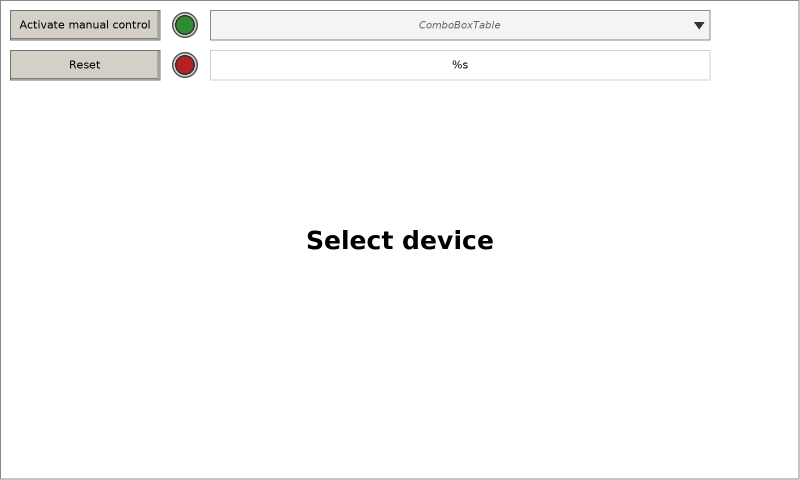
VISUALIZATION ManualControl  // 800x480
VAR_IN_OUT
	fbManualControler	: FB_ManualController ;
	
END_VAR
    Frame (0,0 800x480), input disabled if: fbManualControler.bDisableManualInputs, frame switch variable: fbManualControler.eDevType
        shows VisuUndefinedControl()
        shows VisuValveControl(fbManualControler := fbManualControler)
        shows VisuCylinderControl(fbManualControler := fbManualControler)
        shows VisuAxisControl(fbManualControler := fbManualControler)
        shows VisuPushbuttonLightControl(fbManualControler := fbManualControler)
        shows VisuDigitalInputControl(fbManualControler := fbManualControler)
        shows VisuAnlogInputControl(fbManualControler := fbManualControler)
        shows VisuDigitalOutControl(fbManualControler := fbManualControler)
        shows VisuAnalogOutControl(fbManualControler := fbManualControler)
        shows VisuPWMControl(fbManualControler := fbManualControler)
        shows VisuDoublePWMControl(fbManualControler := fbManualControler)
        shows VisuEncoderInput(fbManualControler := fbManualControler)
        shows VisuAnalogAxisControl(fbManualControler := fbManualControler)
        shows VisuTwoVelocityAxisControl(fbManualControler := fbManualControler)
        shows VisuKL5151Control(fbManualControler := fbManualControler)
        shows VisuKL15XXControl(fbManualControler := fbManualControler)
    Button (10,10 150x30), "Activate manual control", pressed state: fbManualControler.bManualActive
        toggle fbManualControler.bManualActive
    Lamp1 (170,50 30x30), tooltip "component fault active", variable: fbManualControler.bErroractive, style: Lamp-Lamp1-Red
    Lamp1 (170,10 30x30), tooltip "Manual control active", variable: fbManualControler.bManual, style: Lamp-Lamp1-Green
    Textfield (210,50 500x30), "%s", text variable: fbManualControler.sDeviceState
    Button (10,50 150x30), "Reset"
        tap fbManualControler.bReset
    ComboBoxTable (210,10 500x30), variable: fbManualControler.nCmdLookupindex, data array: fbManualControler.arDeviceArray
        p1128707560: fbManualControler.nNumberOfDevices
        p3854506369: fbManualControler.arDeviceArray[INDEX].sName
        p1892666644: fbManualControler.arDeviceArray[INDEX].sType
        p338671338: fbManualControler.arDeviceArray[INDEX].pFunction^
END_VISUALIZATION

// ---- Screens/Manual/toManualButton.TcVIS
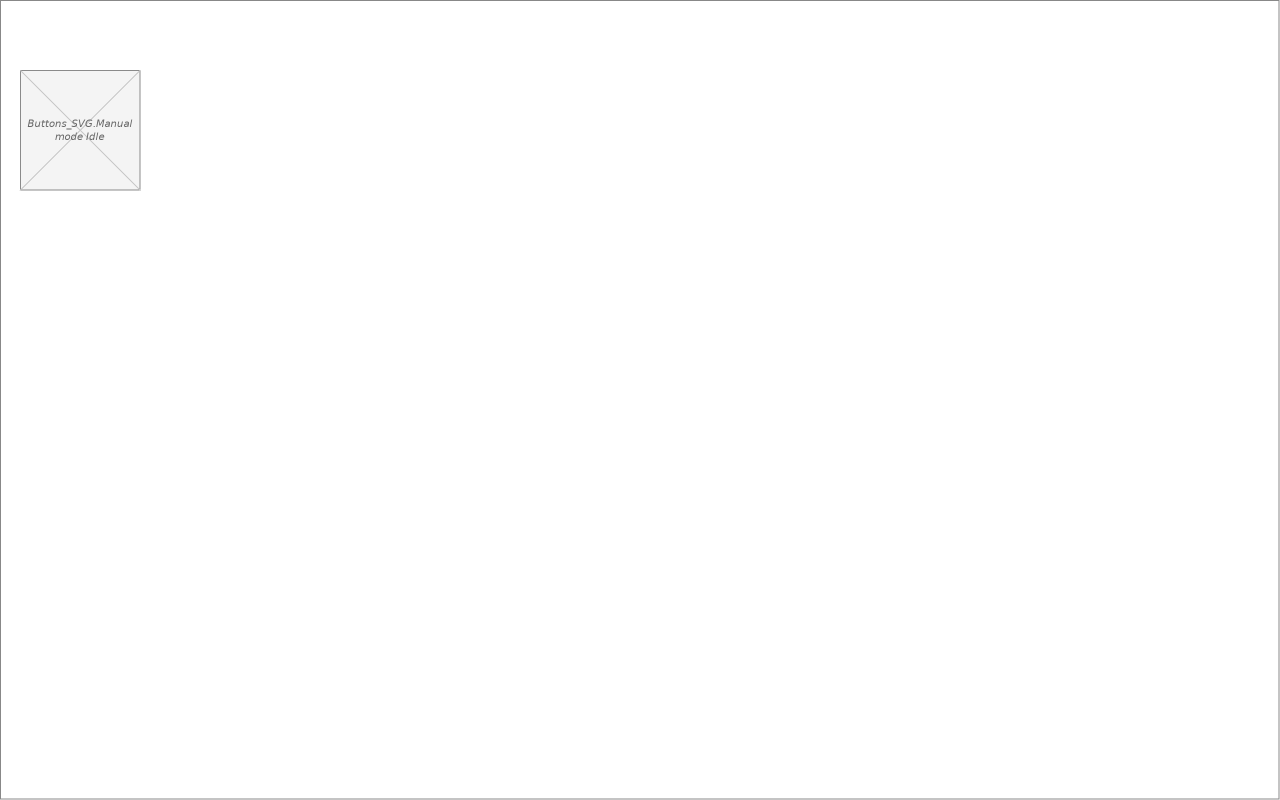
VISUALIZATION toManualButton  // 1280x800
    Image (20,70 120x120), image: Buttons_SVG.Manual mode Idle
        OnMouseClick: toggle GVL_HMI.bCmdManual
END_VISUALIZATION

// ---- Screens/Parameter/ParameterControl.TcVIS
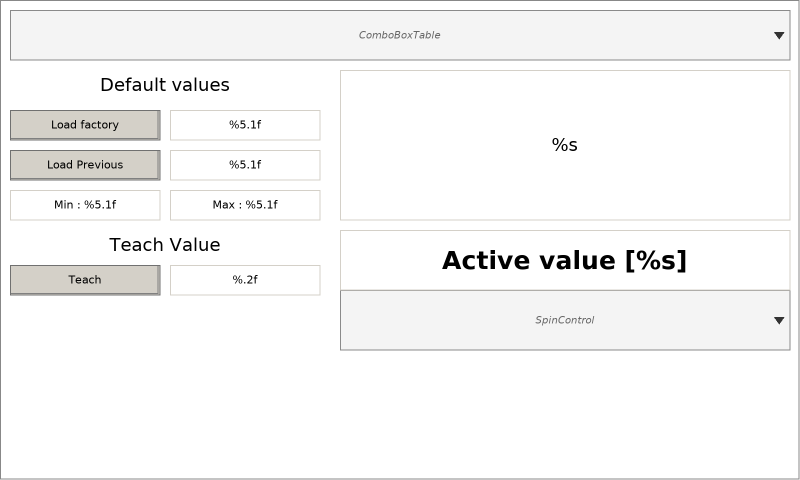
VISUALIZATION ParameterControl  // 800x480
    ComboBoxTable (10,10 780x50), variable: GVL_Parameters.fbParameterHandler.nLookupIndex, data array: GVL_Parameters.fbParameterHandler.arParameters
        p1128707560: GVL_Parameters.fbParameterHandler.nNumberOfParameters
        p3854506369: GVL_Parameters.fbParameterHandler.arParameters[INDEX].nNumber
        p1892666644: GVL_Parameters.fbParameterHandler.arParameters[INDEX].sName
        p338671338: GVL_Parameters.fbParameterHandler.arParameters[INDEX].sType
        p2170511999: GVL_Parameters.fbParameterHandler.arParameters[INDEX].pParameter^
    Group (10,70 310x150)
        Button (0,40 150x30), "Load factory"
            tap GVL_Parameters.fbParameterHandler.bCmdLoadfactory
        Label (0,0 310x30), "Default values"
        Textfield (160,40 150x30), "%5.1f", text variable: GVL_Parameters.fbParameterHandler.arParameters[GVL_Parameters.fbParameterHandler.nLookupIndex].pParameter^.fFactory
            OnMouseClick: write the text variable via VisuDialogs.Numpad, min GVL_Parameters.fbParameterHandler.arParameters[GVL_Parameters.fbParameterHandler.nLookupIndex].pParameter^.fMinimum, max GVL_Parameters.fbParameterHandler.arParameters[GVL_Parameters.fbParameterHandler.nLookupIndex].pParameter^.fMaximum
        Button (0,80 150x30), "Load Previous"
            tap GVL_Parameters.fbParameterHandler.bCmdLoadFromPrevious
        Textfield (160,80 150x30), "%5.1f", text variable: GVL_Parameters.fbParameterHandler.arParameters[GVL_Parameters.fbParameterHandler.nLookupIndex].pParameter^.fSaved
        Textfield (160,120 150x30), "Max : %5.1f", text variable: GVL_Parameters.fbParameterHandler.arParameters[GVL_Parameters.fbParameterHandler.nLookupIndex].pParameter^.fMaximum
            OnMouseClick: write the text variable via VisuDialogs.Numpad
        Textfield (0,120 150x30), "Min : %5.1f", text variable: GVL_Parameters.fbParameterHandler.arParameters[GVL_Parameters.fbParameterHandler.nLookupIndex].pParameter^.fMinimum
            OnMouseClick: write the text variable via VisuDialogs.Numpad
    Textfield (340,70 450x150), "%s", text variable: GVL_Parameters.fbParameterHandler.arParameters[GVL_Parameters.fbParameterHandler.nLookupIndex].pParameter^.sDiscription
    SpinControl (340,290 450x60), variable: GVL_Parameters.fbParameterHandler.arParameters[GVL_Parameters.fbParameterHandler.nLookupIndex].pParameter^.fValue
        p576042468: GVL_Parameters.fbParameterHandler.arParameters[GVL_Parameters.fbParameterHandler.nLookupIndex].pParameter^.fMinimum
        p651134158: GVL_Parameters.fbParameterHandler.arParameters[GVL_Parameters.fbParameterHandler.nLookupIndex].pParameter^.fMaximum
        OnMouseClick: write the text variable via VisuDialogs.Numpad, min GVL_Parameters.fbParameterHandler.arParameters[GVL_Parameters.fbParameterHandler.nLookupIndex].pParameter^.fMinimum, max GVL_Parameters.fbParameterHandler.arParameters[GVL_Parameters.fbParameterHandler.nLookupIndex].pParameter^.fMaximum
    Textfield (340,230 450x60), "Active value [%s]", text variable: GVL_Parameters.fbParameterHandler.arParameters[GVL_Parameters.fbParameterHandler.nLookupIndex].pParameter^.sUnit
    Group (10,230 310x65)
        Label (0,0 310x30), "Teach Value"
        Textfield (160,35 150x30), "%.2f", text variable: GVL_Parameters.fbParameterHandler.arParameters[GVL_Parameters.fbParameterHandler.nLookupIndex].pParameter^.fPrepared
        Button (0,35 150x30), "Teach"
            tap GVL_Parameters.fbParameterHandler.bCmdAcceptTeach
END_VISUALIZATION

// ---- Screens/Parameter/ParButton_PNG.TcVIS
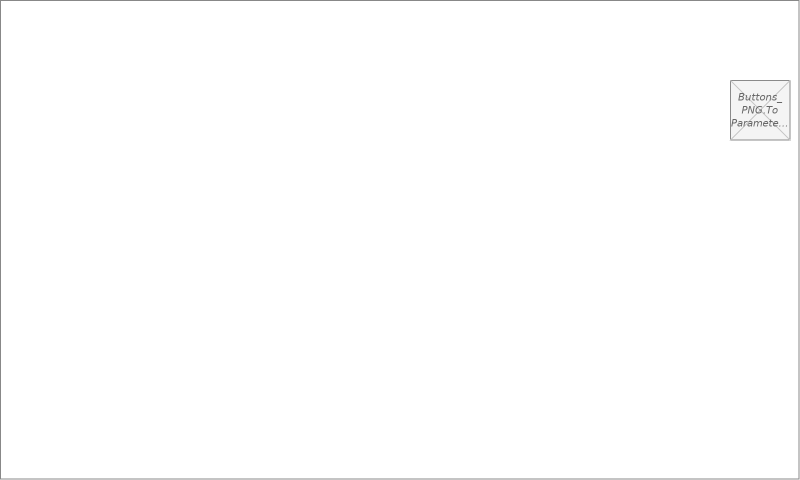
VISUALIZATION ParButton_PNG  // 800x480
VAR_IN_OUT
	bCmdParameter	: BOOL ; // to parameter screen
END_VAR
    Image (730,80 60x60), image: Buttons_PNG.To Parameter Screen
        OnMouseClick: toggle bCmdParameter
END_VISUALIZATION

// ---- Screens/Startup Screen/LogoScreen_PNG.TcVIS
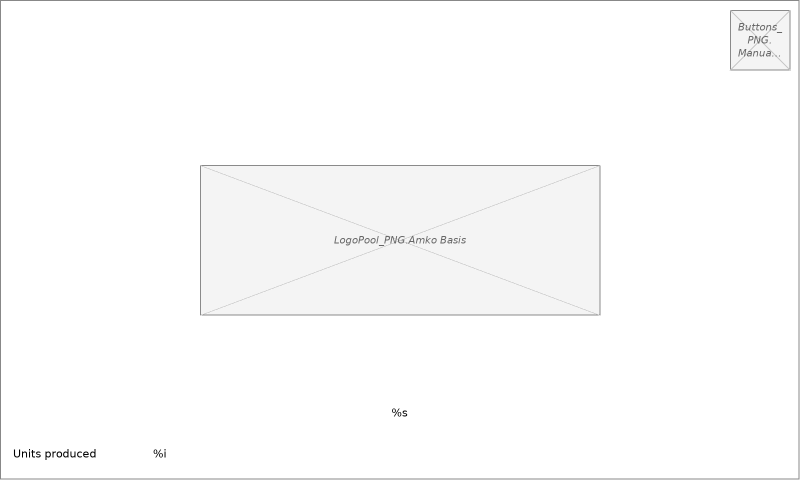
VISUALIZATION LogoScreen_PNG  // 800x480
VAR_INPUT
	nUnitsProduced	: UDINT; // HMI Main total units produced
END_VAR
VAR_IN_OUT
	bCmdManual		: BOOL ; // HMI switch to manual mode
END_VAR
    Frame (0,0 800x480)
        shows ManualButton_PNG(bCmdManual := bCmdManual)
    Image (200,165 400x150), image: LogoPool_PNG.Amko Basis
    Textfield (183,404 433x18), "%s", tooltip "Operator messagages", text variable: GVL_Message.sOPeratorMessage
    Textfield (110,439 100x30), "%i", text variable: nUnitsProduced
    Label (10,439 100x30), "Units produced"
END_VISUALIZATION

// ---- Screens/Startup Screen/LogoScreenBliss_PNG.TcVIS
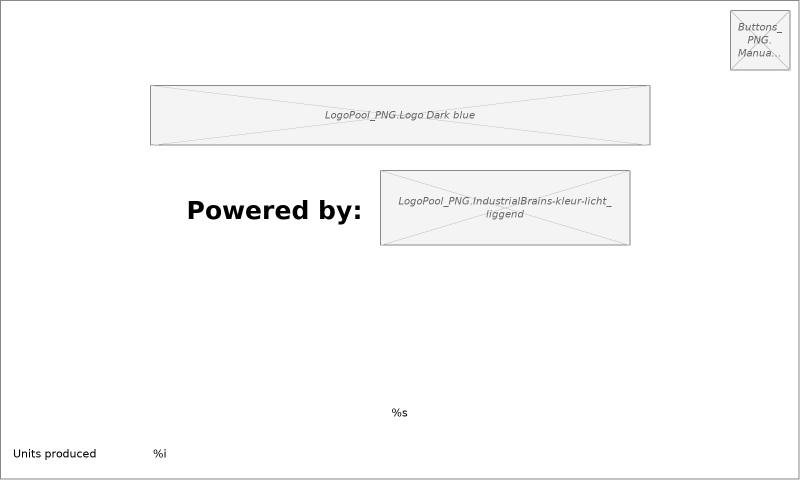
VISUALIZATION LogoScreenBliss_PNG  // 800x480
VAR_INPUT
	nUnitsProduced	: UDINT; // HMI Main total units produced
END_VAR
VAR_IN_OUT
	bCmdManual		: BOOL ; // HMI switch to manual mode
END_VAR
    Frame (0,0 800x480)
        shows ManualButton_PNG(bCmdManual := bCmdManual)
    Image (150,85 500x60), image: LogoPool_PNG.Logo Dark blue
    Image (380,170 250x75), image: LogoPool_PNG.IndustrialBrains-kleur-licht_liggend
    Textfield (183,404 433x18), "%s", tooltip "Operator messagages", text variable: GVL_Message.sOPeratorMessage
    Textfield (110,439 100x30), "%i", text variable: nUnitsProduced
    Label (10,439 100x30), "Units produced"
    Label (179,150 200x120), "Powered by:"
END_VISUALIZATION

// ---- Screens/Startup Screen/LogoScreen_SVG.TcVIS
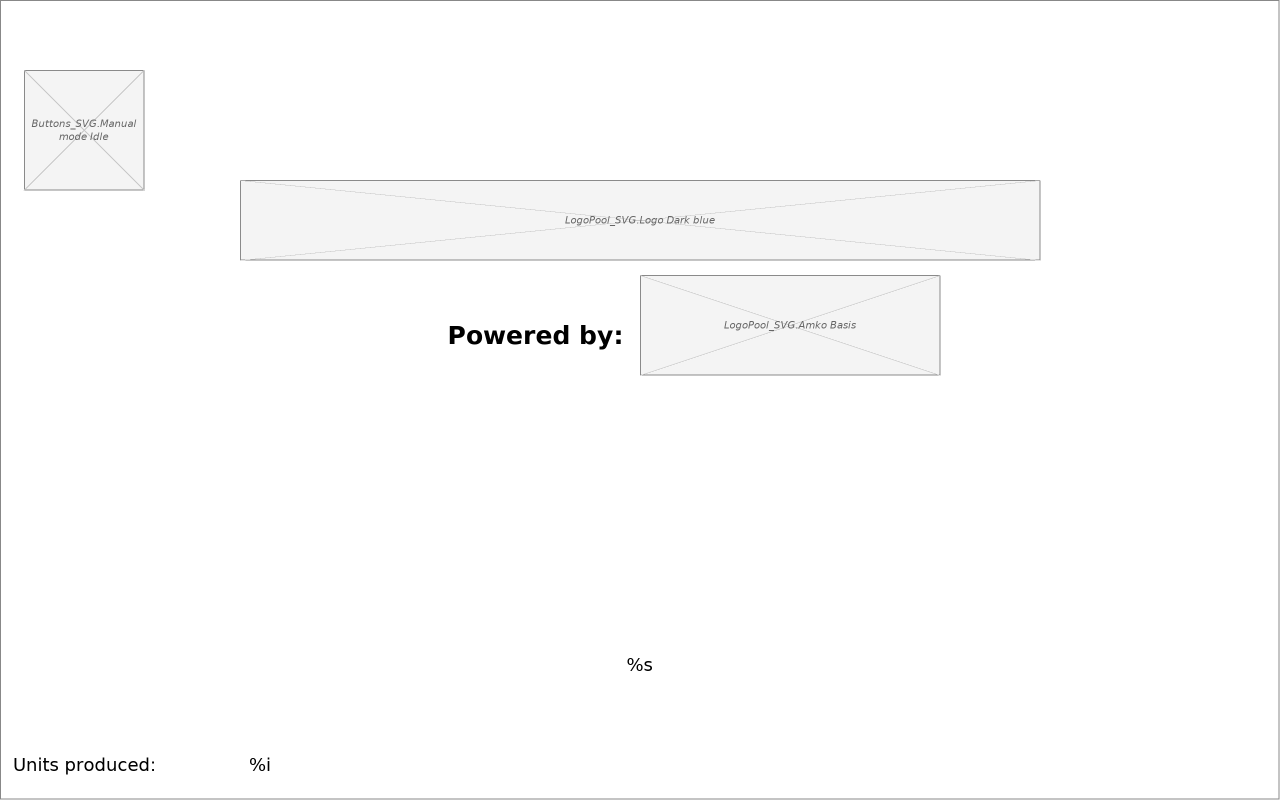
VISUALIZATION LogoScreen_SVG  // 1280x800
VAR_IN_OUT
	nUnitsProduced : UDINT ; // Units produced in machine lifetime
END_VAR
    Frame (4,0 1280x800)
        shows toManualButton()
    Image (240,180 800x80), image: LogoPool_SVG.Logo Dark blue
    Image (640,275 300x100), image: LogoPool_SVG.Amko Basis
    Label (440,275 200x120), "Powered by:"
    Textfield (240,650 800x30), "%s", tooltip "Operator messagages", text variable: GVL_Message.sOPeratorMessage
    Textfield (160,750 200x30), "%i", text variable: nUnitsProduced
    Label (10,750 150x30), "Units produced:"
END_VISUALIZATION

// ---- Screens/Startup Screen/LogoScreenBlanc_SVG.TcVIS
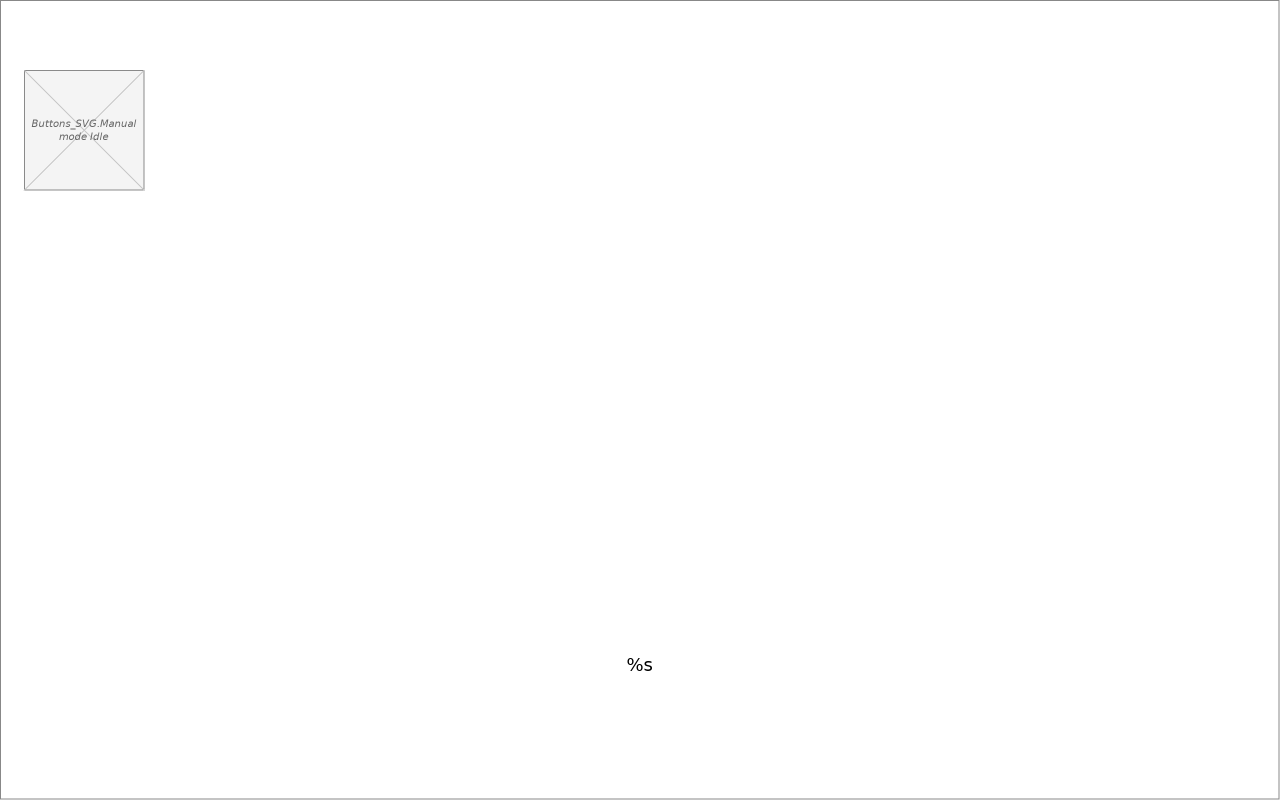
VISUALIZATION LogoScreenBlanc_SVG  // 1280x800
    Frame (4,0 1280x800)
        shows toManualButton()
    Textfield (240,650 800x30), "%s", tooltip "Operator messagages", text variable: GVL_Message.sOPeratorMessage
END_VISUALIZATION

// ---- Screens/State_PNG/Idle_PNG.TcVIS
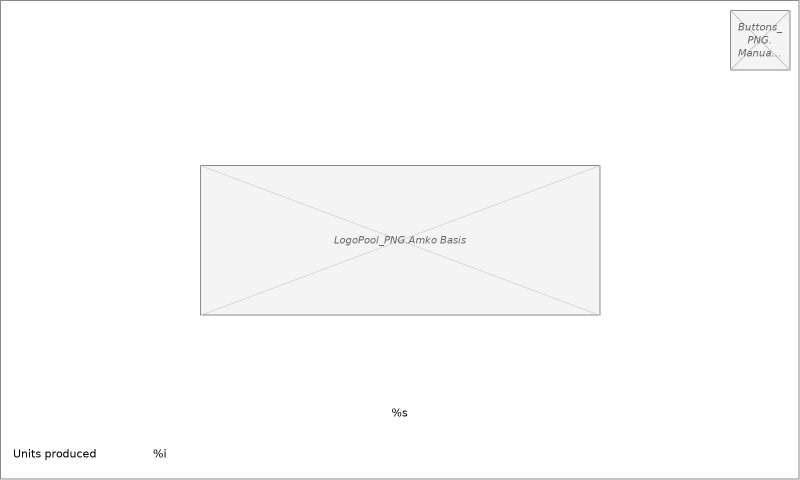
VISUALIZATION Idle_PNG  // 800x480
VAR_IN_OUT
	nUnitsProduced	: UDINT ;
END_VAR
    Frame (0,0 800x480)
        shows LogoScreen_PNG(nUnitsProduced := nUnitsProduced, bCmdManual := GVL_HMI.bCmdManual)
END_VISUALIZATION

// ---- Screens/State_PNG/Manual_PNG.TcVIS
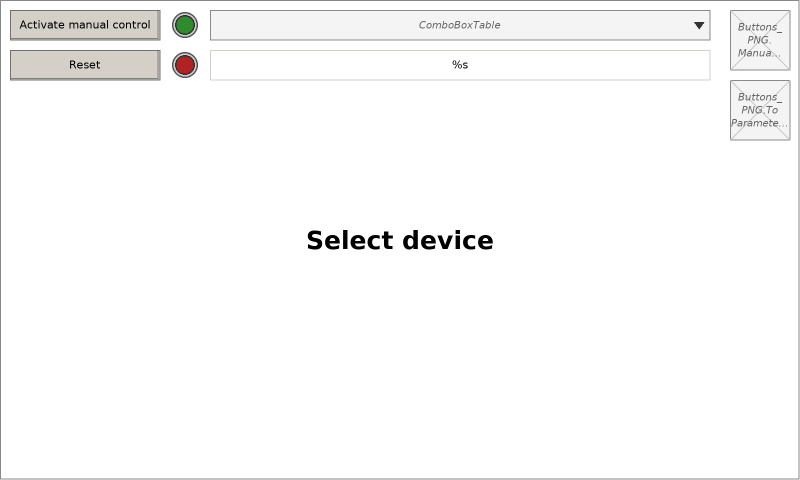
VISUALIZATION Manual_PNG  // 800x480
VAR_IN_OUT
	bCmdManual  	: BOOL ; // switch to manual screen
	bCmdParameter	: BOOL ; // switch to parameter screen
END_VAR
    Frame (0,0 800x480)
        shows ManualControl(fbManualControler := Device_Library.GVL_DevManual.fbManualControler)
    Frame (0,0 800x480)
        shows ManualButton_PNG(bCmdManual := bCmdManual)
    Frame (0,0 800x480)
        shows ParButton_PNG(bCmdParameter := bCmdParameter)
END_VISUALIZATION

// ---- Screens/State_PNG/Parameter_PNG.TcVIS
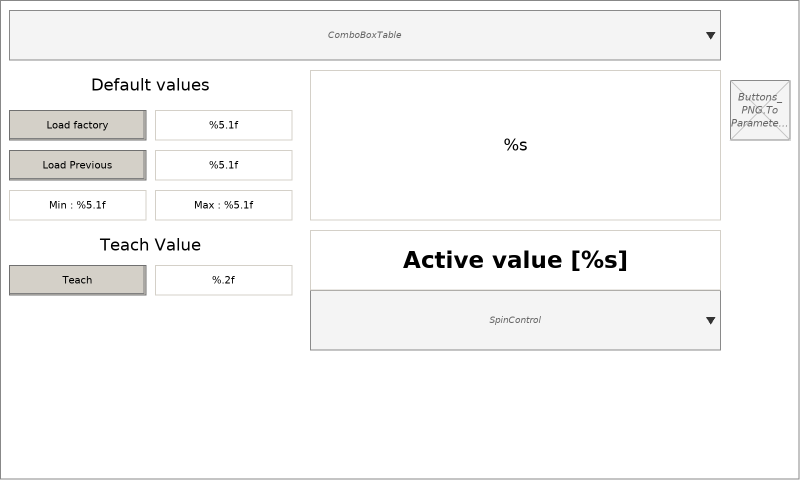
VISUALIZATION Parameter_PNG  // 800x480
VAR_IN_OUT
	bCmdParameter : BOOL ; // Return from parameter screen
END_VAR
    Frame (0,0 800x480)
        shows ParButton_PNG(bCmdParameter := bCmdParameter)
    Frame (0,0 730x480)
        shows ParameterControl()
END_VISUALIZATION

// ---- Screens/State_PNG/Settings_PNG.TcVIS
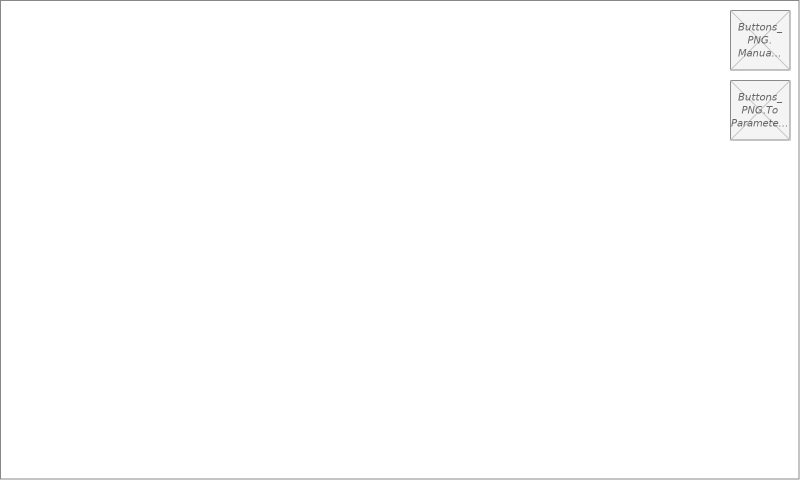
VISUALIZATION Settings_PNG  // 800x480
    Frame (0,0 800x480)
        shows ManualButton_PNG(bCmdManual := GVL_HMI.bCmdManual)
    Frame (0,0 800x480)
        shows ParButton_PNG(bCmdParameter := GVL_HMI.bCmdParemeter)
END_VISUALIZATION

// ---- Screens/State_SVG/Manual.TcVIS
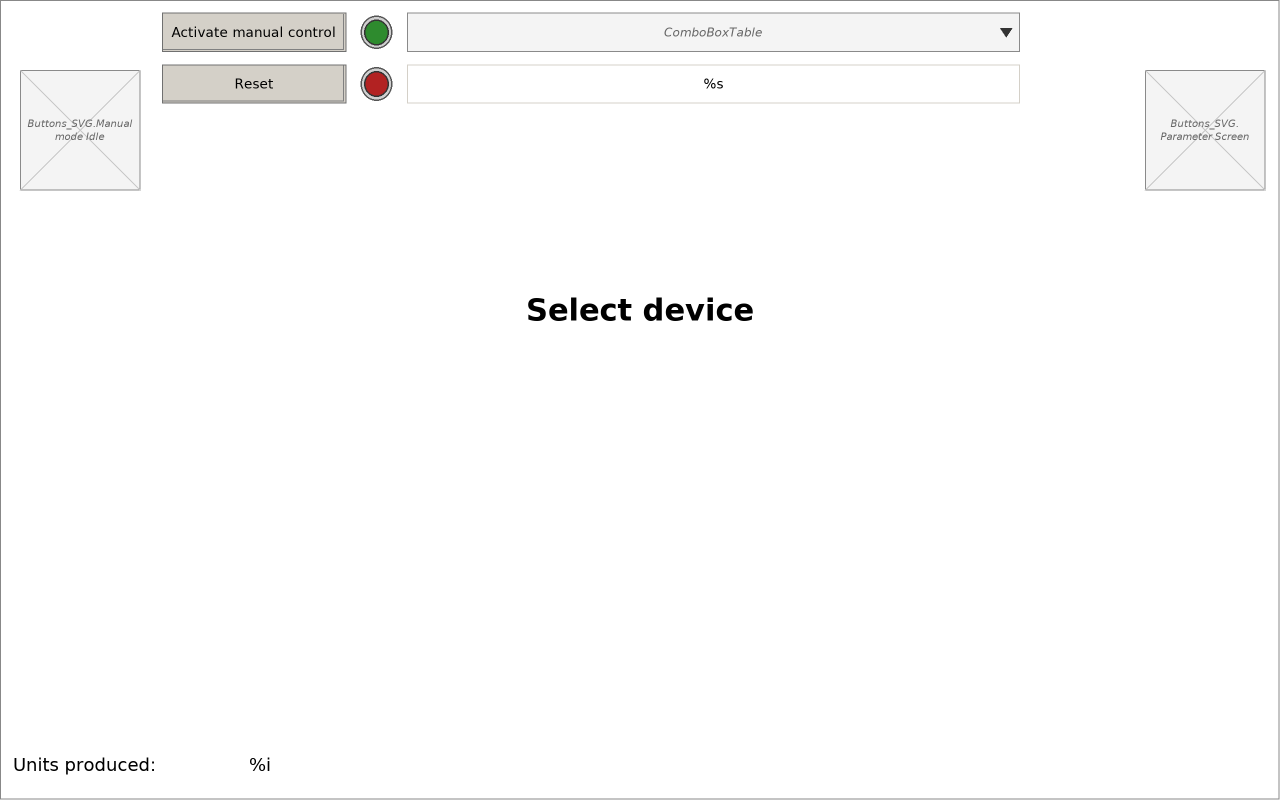
VISUALIZATION Manual  // 1280x800
VAR_IN_OUT
	bCmdParameter : BOOL ;
	nUnitsProduced : UDINT ; // Units produced in machine lifetime
END_VAR
    Frame (0,0 1280x800)
        shows toManualButton()
    Frame (0,0 1280x800)
        shows Settings(bCmdParameter := bCmdParameter, nUnitsProduced := nUnitsProduced)
    Frame (150,0 980x620)
        shows ManualControl(fbManualControler := Device_Library.GVL_DevManual.fbManualControler)
END_VISUALIZATION

// ---- Screens/State_SVG/ParameterScreen.TcVIS
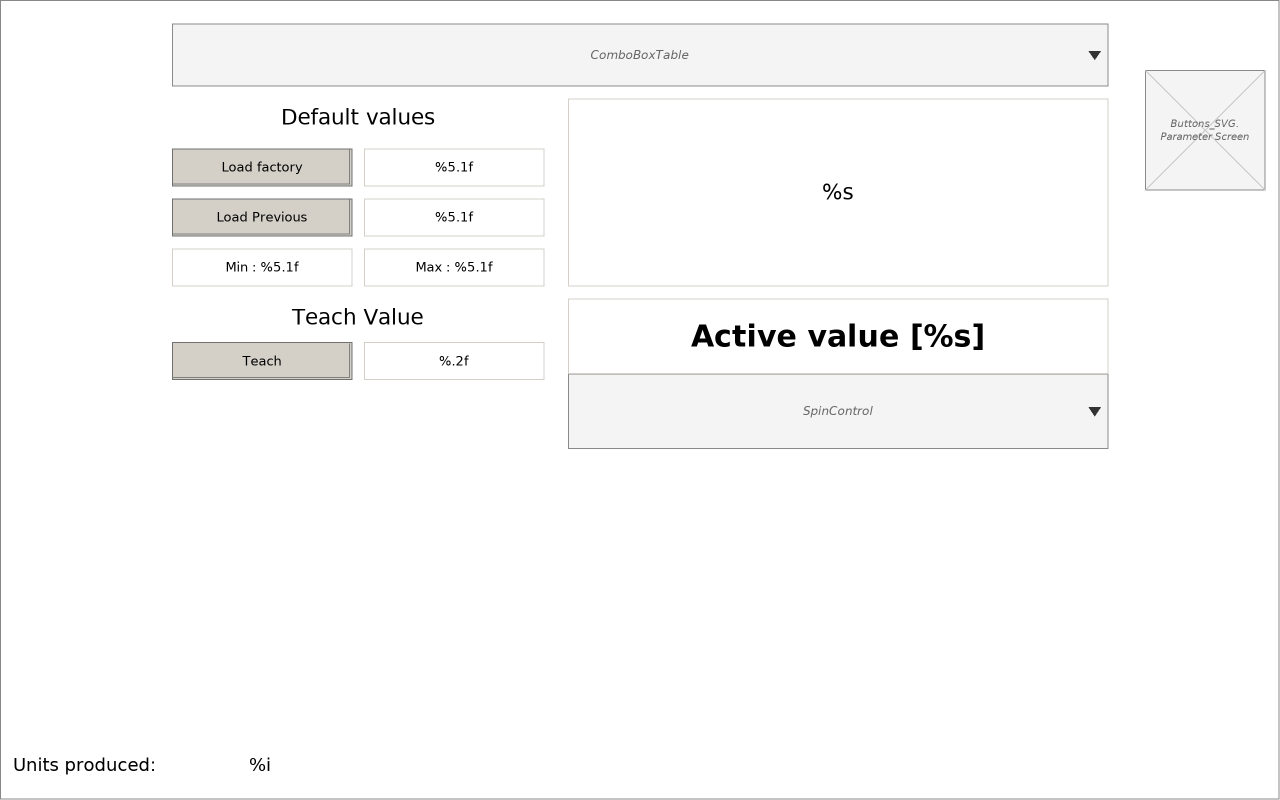
VISUALIZATION ParameterScreen  // 1280x800, background image BackGroundImagePool_SVG.Background_Sides
VAR_IN_OUT
	bCmdParameter : BOOL ; // Go to parameter screen
	nUnitsProduced : UDINT ; // Units produced in machine lifetime
END_VAR
    Frame (0,0 1280x800)
        shows Settings(bCmdParameter := bCmdParameter, nUnitsProduced := nUnitsProduced)
    Frame (160,11 960x600)
        shows ParameterControl()
END_VISUALIZATION

// ---- Screens/State_SVG/Settings.TcVIS
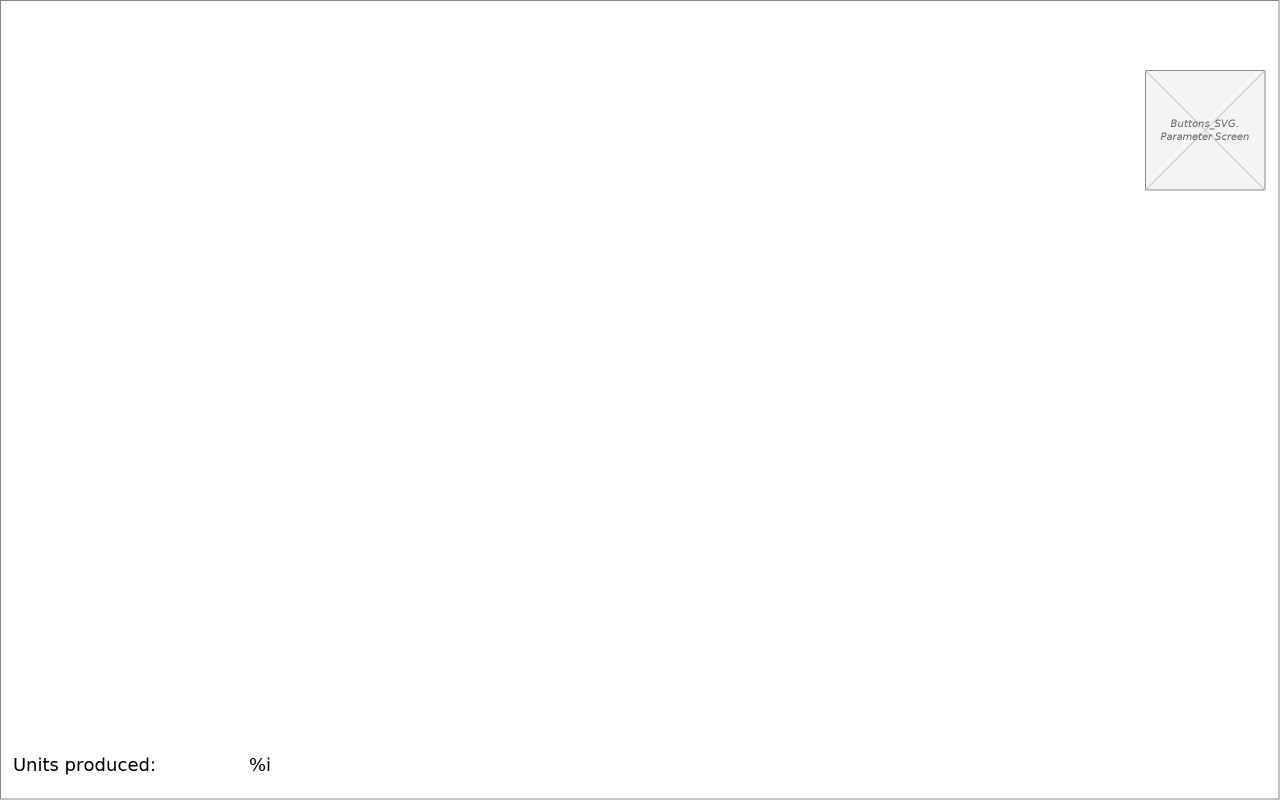
VISUALIZATION Settings  // 1280x800
VAR_IN_OUT
	bCmdParameter : BOOL ; // Go to parameter screen
	nUnitsProduced : UDINT ; // Units produced in machine lifetime
END_VAR
    Label (10,750 150x30), "Units produced:"
    Textfield (160,750 200x30), "%i", text variable: nUnitsProduced
    Image (1145,70 120x120), image: Buttons_SVG.Parameter Screen
        OnMouseClick: toggle bCmdParameter
        OnMouseClick: VisuUserMgmt Type=Login
END_VISUALIZATION

// ---- Screens/State_SVG/Idle.TcVIS
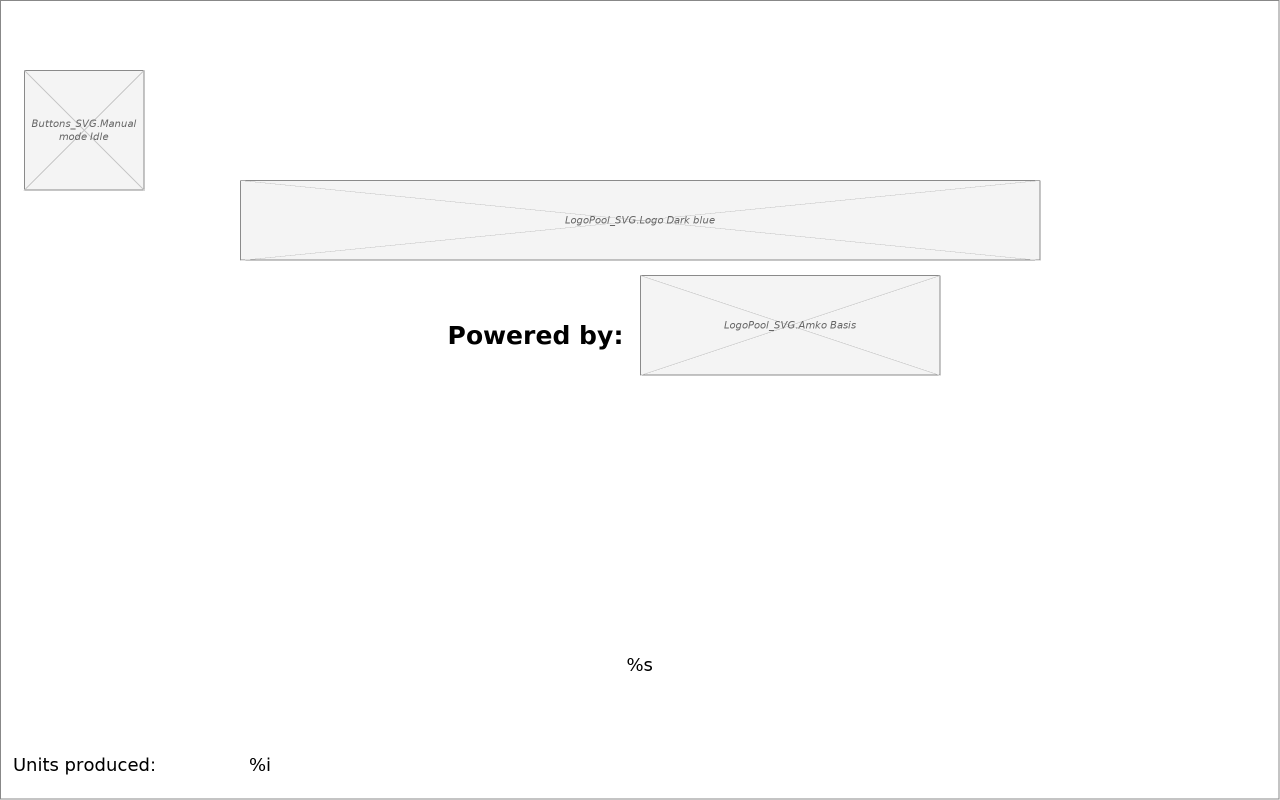
VISUALIZATION Idle  // 1280x800
VAR_IN_OUT
	nUnitsProduced : UDINT ; // Units produced in machine lifetime
END_VAR
    Frame (0,0 1280x800), frame switch variable: 0
        shows LogoScreen_SVG(nUnitsProduced := nUnitsProduced)
        shows Settings()
        shows ParameterScreen()
        shows Run()
END_VISUALIZATION

// ---- TextLists/E_ComponentTypes.TcTLO
TEXTLIST E_ComponentTypes
  0 = 'NA'
  10 = 'Cylinder'
  11 = 'Axis'
  20 = 'EstopButton'
  21 = 'EstopBumper'
  22 = 'Pushbutton'
  23 = 'Switch'
  30 = 'SafeIO'
  31 = 'Rio_Box'
  32 = 'Rio_Slot'
  33 = 'Encoder'
  34 = 'DiSensor'
  40 = 'ServoDrive'
  50 = 'HMI'
  51 = 'RemoteOS'
  52 = 'RemoteDB'
  60 = 'Assembly'
  61 = 'SubAssembly'
  100 = 'MainProgram'
  101 = 'StepProgram'
  102 = 'FunctionBlock'
   = ''
END_TEXTLIST

// ---- TextLists/E_FaultTypes.TcTLO
TEXTLIST E_FaultTypes
  0 = 'NA'
  1 = 'OM'
  2 = 'MC'
  3 = 'CF'
  4 = 'FF'
   = ''
END_TEXTLIST

// ---- TextLists/E_Locations.TcTLO
TEXTLIST E_Locations
  0 = 'Main PLC'
  1 = '230V Main supply'
  2 = '24V Main supply'
  3 = 'Main air supply'
  4 = 'Main Screen'
  5 = 'Main IO'
   = ''
END_TEXTLIST

// ---- TextLists/E_MessageNumbers.TcTLO
TEXTLIST E_MessageNumbers
  0 = 'NA_NoMessage'
  1 = 'FF_Unknown'
  2 = 'FF_NoCommunication'
  3 = 'FF_ComunicationFault'
  4 = 'FF_Overload'
  5 = 'FF_EncoderFault'
  6 = 'FF_SlaveFault'
  7 = 'FF_AxisFault'
  8 = 'FF_DriveFault'
  9 = 'FF_Collision'
  100 = 'CF_FeedbackFault'
  101 = 'CF_WrongDirection'
  102 = 'CF_MoveToFast'
  103 = 'CF_MoveToSlow'
  104 = 'CF_WrongPosition'
  105 = 'CF_Obstruction'
  200 = 'MC_WaitingForproduct'
  201 = 'MC_WaitingForOperator'
  202 = 'MC_WaitingForModule'
  203 = 'MC_WaitingForMaster'
  204 = 'MC_WaitingForSlave'
  205 = 'MC_WrongPosition'
  300 = 'OM_AlmostEmpty'
  301 = 'OM_Finished'
  302 = 'OM_ready'
  900 = 'FF_MessageTest'
  901 = 'CF_MessageTest'
  902 = 'MC_MessageTest'
  903 = 'OM_MessageTest'
   = ''
END_TEXTLIST

// ---- TextLists/E_ParameterNames.TcTLO
TEXTLIST E_ParameterNames
  0 = 'Mpar_StitchLengthLong'
  1 = 'MPar_StitchLengthShort'
  2 = 'MPar_MaxSpeed'
  3 = 'Mpar_MinSpeed'
  4 = 'Mpar_ManualMaxSpeed'
  5 = 'Mpar_BacktackSpeed'
  6 = 'Mpar_SlowEndSpeed'
  7 = 'Mpar_HomingSpeed'
  8 = 'Mpar_CuttingSpeed'
  9 = 'Mpar_MaxAcceleration'
  10 = 'Mpar_MaxDeceleration'
  11 = 'Mpar_Jerk'
  12 = 'Mpar_BacktackAcceleration'
  13 = 'Mpar_BacktackDeceleration'
  14 = 'Mpar_TransferAcceleration'
  15 = 'Mpar_TransferDeceleration'
  16 = 'Mpar_CylinderTimeoutMargin'
  17 = 'Cpar_NeedleSensorPos'
  18 = 'Cpar_NeedlePosUp'
  19 = 'Cpar_NeedlePosInMaterial'
  20 = 'Cpar_NeedleposDown'
  21 = 'Cpar_NeedlePosStartCut'
  22 = 'Cpar_NeedlePosStopCut'
  23 = 'Cpar_NeedlePosEndCut'
  24 = 'Cpar_NeedlePosRelTensCut'
  25 = 'Cpar_NeedlePosHoldThread'
  26 = 'Cpar_NeedlePosStartRelTension'
  27 = 'Cpar_NeedlePosStopRelTension'
  28 = 'Cpar_NeedlePosChangeDirUp'
  29 = 'Cpar_NeedlePosClearStart'
  30 = 'Cpar_NeedlePosClearEnd'
  31 = 'Cpar_NeedlePosRef'
  32 = 'Cpar_NeedlePosPause'
  33 = 'Cpar_SensorPreEdgeDetDistance'
  34 = 'Cpar_sensorEdgeDetDistance'
  35 = 'Opar_NeedleSensorPos'
  36 = 'Opar_NeedlePosUp'
  37 = 'Opar_NeedlePosInMaterial'
  38 = 'Opar_NeedleposDown'
  39 = 'Opar_NeedlePosStartCut'
  40 = 'Opar_NeedlePosStopCut'
  41 = 'Opar_NeedlePosEndCut'
  42 = 'Opar_NeedlePosRelTensCut'
  43 = 'Opar_NeedlePosHoldThread'
  44 = 'Opar_NeedlePosStartRelTension'
  45 = 'Opar_NeedlePosStopRelTension'
  46 = 'Opar_NeedlePosChangeDir'
  47 = 'Opar_NeedlePosClearStart'
  48 = 'Opar_NeedlePosClearEnd'
  49 = 'Opar_NeedlePosPause'
  50 = 'Ppar_BacktackStitchStartFwd'
  51 = 'Ppar_BacktackStitchStartRev'
  52 = 'Ppar_BacktackStitchEndFwd'
  53 = 'Ppar_BacktackStitchEndRev'
  54 = 'Ppar_AutomaticSpeed'
  55 = 'Ppar_StitchStretch'
  56 = 'Ppar_ThreadLengthAdition'
  57 = 'Ppar_ThreadBreakDelay'
  58 = 'Mpar_MaxVelocity'
  59 = 'Mpar_MinVelocity'
  60 = 'Mpar_ManualMaxVelocity'
  61 = 'Mpar_MLTMaxAcceleration'
  62 = 'Mpar_MLTMaxDeceleration'
  63 = 'Mpar_TraverseLength'
  64 = 'Mpar_CylTimeOutMargine'
  65 = 'Mpar_HomingVelocity'
  66 = 'Mpar_SewingcartLength'
  67 = 'Mpar_ClampCartLength'
  68 = 'Mpar_MaxClampCartVelocity'
  69 = 'Mpar_TraverseReturnVelocity'
  70 = 'Mpar_ToStartvelocity'
  71 = 'Mpar_InspectionDistance'
  72 = 'Cpar_PosHoming'
  73 = 'Cpar_PosSuportCyl_1'
  74 = 'Cpar_PosSuportCyl_2'
  75 = 'Cpar_PosSuportCyl_3'
  76 = 'Cpar_PosService'
  77 = 'Cpar_PosBobinChange'
  78 = 'Cpar_PosEnd'
  79 = 'Cpar_TimeBaseClampsClose'
  80 = 'Cpar_TimeBaseClampsRel'
  81 = 'Cpar_TimeCartClampsClose'
  82 = 'Cpar_TimeCartClampsRel'
  83 = 'Cpar_TimeCartBrakeApply'
  84 = 'Cpar_TimeCartBrakeRel'
  85 = 'Cpar_TimeSupportExp_1'
  86 = 'Cpar_TimeSupportRet_1'
  87 = 'Cpar_TimeSupportExp_2'
  88 = 'Cpar_TimeSupportRet_2'
  89 = 'Cpar_TimeSupportExp_3'
  90 = 'Cpar_TimeSupportRet_3'
  91 = 'Cpar_TimeBobinPlateClose'
  92 = 'Cpar_TimeBobinPlateOpen'
  93 = 'Cpar_PosFlagSewingcart'
  94 = 'Cpar_PosSensorClampCart'
  95 = 'Cpar_SupportCylWidth'
  96 = 'Cpar_ClampCartFlagWidth'
  97 = 'Cpar_PosMaterialStart'
  98 = 'Opar_HomePosition'
  99 = 'Opar_PosSuportCyl_1'
  100 = 'Opar_PosSuportCyl_2'
  101 = 'Opar_PosSuportCyl_3'
  102 = 'Opar_PosService'
  103 = 'Opar_PosBobinChange'
  104 = 'Opar_PosEnd'
  105 = 'Opar_PosMatStart'
  106 = 'Ppar_ProductLenght'
  107 = 'Ppar_ProductStretch'
  108 = 'Ppar_StartStretchFactor'
  109 = 'Ppar_StartStretchLength'
  110 = 'Ppar_ReverseStretch'
  111 = 'Ppar_MatBlowDistance'
   = ''
END_TEXTLIST

// ---- TextLists/GlobalTextList.TcGTLO
TEXTLIST GlobalTextList
  0 = ' Act velocity:'
  268 = '%.2f'
  923 = '%5.1f'
  237 = '%5.2f'
  222 = '%f'
  909 = '%f.1'
  388 = '%i'
  568 = '%n'
  596 = '%s'
  864 = '%S'
  555 = '123456789'
  560 = 'Accept'
  869 = 'Accept change'
  196 = 'Act velocity'
  224 = 'Activate manual control'
  791 = 'Active value'
  638 = 'Active value [%s]'
  505 = 'ActiveValue'
  584 = 'Actual Position:'
  252 = 'Actual velocity:'
  62 = 'Administrator'
  146 = 'AutpotVelo:'
  614 = 'CCW'
  447 = 'CCW Fast'
  633 = 'Clock Wise'
  167 = 'Clock wise Fast'
  50 = 'Close'
  96 = 'Clounter clock wise Fast'
  825 = 'Command distance:'
  263 = 'Command Position:'
  851 = 'Command velocity:'
  1 = 'component fault active'
  52 = 'CounterClockWise'
  641 = 'CW'
  297 = 'CW Fast'
  626 = 'Cycle Time [ms]'
  264 = 'Default values'
  175 = 'device initialized'
  364 = 'Discription'
  740 = 'Duty cycle [%]'
  932 = 'Fault Messages'
  391 = 'FF'
  952 = 'Functionblock'
  660 = 'Hardware Movement completion time is lower then minimum'
  274 = 'Home'
  546 = 'Input value: %i'
  879 = 'Jog Forward'
  223 = 'Jog Inching'
  370 = 'Jog reverse'
  739 = 'Label'
  7 = 'Light blink fast'
  137 = 'Light blink slow'
  679 = 'Light off'
  616 = 'Light On'
  154 = 'Load factory'
  624 = 'Load Previous'
  291 = 'Location'
  145 = 'Login'
  58 = 'LogOut'
  804 = 'Manual control active'
  278 = 'Max : %5.1f'
  111 = 'Maximum'
  796 = 'Maxuimum : %5.1f'
  520 = 'Min : %5.1f'
  272 = 'Min: %5.1f'
  936 = 'Minimum : %5.1f'
  948 = 'Move to target position'
  356 = 'Moving:'
  298 = 'None'
  11 = 'Number'
  313 = 'ON'
  463 = 'Open'
  293 = 'Operator'
  204 = 'Operator messagages'
  425 = 'Output A'
  527 = 'Output A on'
  808 = 'Output B'
  110 = 'Output B On'
  39 = 'Output value:'
  417 = 'Powe:red by '
  898 = 'Powered by '
  482 = 'Powered by: '
  704 = 'Pulse'
  174 = 'Reset'
  488 = 'RESET'
  458 = 'RESET FAULTS'
  69 = 'Run CCw'
  559 = 'Run CCW'
  658 = 'Run CCW Fast'
  493 = 'Run Clockwise'
  220 = 'Run Clockwise Fast'
  212 = 'Run Counter clockwise'
  691 = 'Run Counter clockwise Fast'
  928 = 'Run CW'
  629 = 'Run CW Fast'
  138 = 'Run CWW'
  400 = 'Select device'
  320 = 'Set Value'
  107 = 'Snooze'
  795 = 'SNOOZE'
  933 = 'support cylinder 3'
  942 = 'TD'
  771 = 'Teach'
  229 = 'Teach Value'
  186 = 'Teach values'
  177 = 'Time'
  553 = 'Time to close [ms]'
  243 = 'Time to open [ms]'
  132 = 'Type'
  389 = 'Under construction'
  576 = 'Units produced'
  855 = 'Units produced:'
  965 = 'Utilities_Library.GVL_Message.arActiveFaults[4].FaultType'
  643 = 'WaitingForProduct'
  528 = 'Weccome'
  246 = 'Welcome'
  730 = 'Welcomekom'
  634 = 'Welkom'
END_TEXTLIST

// ---- TextLists/TL_MessageDiscriptions.TcTLO
TEXTLIST TL_MessageDiscriptions
  0 = 'No message active'
  1 = 'Unknown error occured'
  2 = 'No communication detected'
  3 = 'Communication error detected (does not match expected com)'
  4 = 'Hardware overload detected'
  5 = 'Encoder signal incorrect or not present'
  6 = 'Slave system is has active fatal fault'
  7 = 'Axis fault feedback'
  8 = 'Axis drive fault'
  9 = 'Collision detected between 2 or more parts of the machine'
  100 = 'Hardware feedback is does not match expected'
  101 = 'Hardware moving in incorrect direction'
  102 = 'Hardware movement completion time is lower then minimum'
  103 = 'Hardware movement maximum time was exceeded'
  104 = 'Hardware is at different position then expected'
  105 = 'Obstruction detected in movement path'
  200 = 'Waiting for product'
  201 = 'Waiting for operator action'
  202 = 'Waiting for other module'
  203 = 'Waiting Waiting for master'
  204 = 'Waiting for slave'
  205 = 'Action or command not possible in current position'
  300 = 'Product is almost empty refif is required'
  301 = 'Product or action is finished'
  302 = 'Ready for new task'
  900 = 'Fatal fault message test'
  901 = 'Cycle fault message test'
  902 = 'Missing condition message test'
  903 = 'Operator message test'
   = ''
END_TEXTLIST
